PROGRAM MAIN
VAR
	isFirstStart : BOOL := TRUE;
	// valve_01 : FB_Valve_monostable;
	valve_01 : Valve_mono;
	
END_VAR

// Set IN(IT)
valve_01.MaxOpenCloseDuration := 15;// this setting can be reduced during test without the fysical Valve

IF isFirstStart THEN
	// Init the Valve at startup (for test/demo)
	GVL_VCM.io_values.I_isClosed := TRUE;
END_IF

// Do stuff
valve_01(Valve:= GVL_VCM.valve01, I_O:= GVL_VCM.io_values);

isFirstStart := FALSE;

END_PROGRAM

(* stored: Version 1.1.0.1, ProductVersion 3.1.4024.12
   POU MAIN: Id {617330db-b8e1-492e-94bc-52a923c83901}, SpecialFunc None *)
